(* CODESYS project Uppgift-13.project

Project tree, tasks and I/O mapping:
  Device : CODESYS Control Win V3, 3S - Smart Software Solutions GmbH, order no. 305021, version 3.5.10.40
    application Application
      libraries: Standard, * (System)
      task MainTask (cyclic, interval t#20ms, priority 1) calls PLC_PRG
      program PLC_PRG [SFC]: OpenDoor, ClosingDoor, HooldDoor, HoldLampLight, ResetValues
      global variables GVL
      Symbols
*)

// Device/Application/GVL
{attribute 'qualified_only'}
VAR_GLOBAL
	PushButton: BOOL;
	SensorOpen: BOOL;
	SensorClose: BOOL;
	MotorForward: BOOL;
	MotorReverse: BOOL;
	TopLight: BOOL;
	DOOROPENLOCK: BOOL; // Is used for lock the door open.
	HoldDoorTime: TON;
END_VAR

// Device/Application/PLC_PRG
PROGRAM PLC_PRG
VAR
	HoldDoorTime: TON;
	DoorHoldTimeElipse: TIME;
	DoorHoldTimeElipse2: TIME;
	HoldDoorTimeOff: TOF;
	TON_0: TON;
	TOF_0: TOF;
	Lampsignal: BOOL;
	BlinkingLampsignal: BOOL;
END_VAR
VAR // added by the converter: edge detectors and wires of the graphical bodies
    _w1, _w2, _w3, _w4 : ANY;
END_VAR

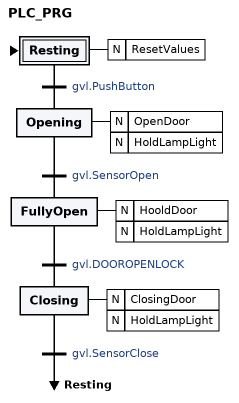
INITIAL_STEP Resting:
    ResetValues(N);
END_STEP
TRANSITION FROM Resting TO Opening
    := gvl.PushButton;
END_TRANSITION
STEP Opening:
    OpenDoor(N);
    HoldLampLight(N);
END_STEP
TRANSITION FROM Opening TO FullyOpen
    := gvl.SensorOpen;
END_TRANSITION
STEP FullyOpen:
    HooldDoor(N);
    HoldLampLight(N);
END_STEP
TRANSITION FROM FullyOpen TO Closing
    := gvl.DOOROPENLOCK;
END_TRANSITION
STEP Closing:
    ClosingDoor(N);
    HoldLampLight(N);
END_STEP
TRANSITION FROM Closing TO Resting
    := gvl.SensorClose;
END_TRANSITION

ACTION OpenDoor:
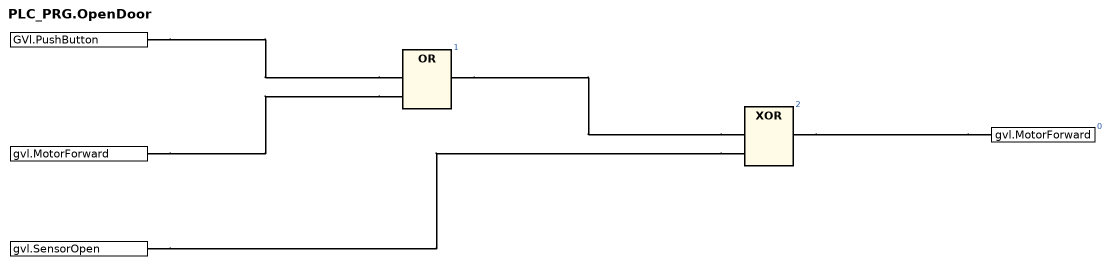
gvl.MotorForward := _w1;
_w1 := (GVl.PushButton OR gvl.MotorForward) XOR gvl.SensorOpen;
END_ACTION

ACTION ClosingDoor:
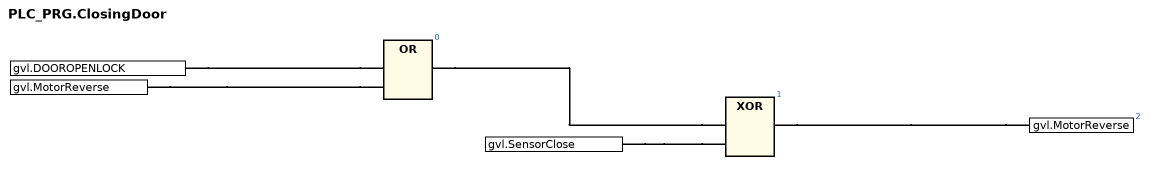
gvl.MotorReverse := (gvl.DOOROPENLOCK OR gvl.MotorReverse) XOR gvl.SensorClose;
END_ACTION

ACTION HooldDoor:
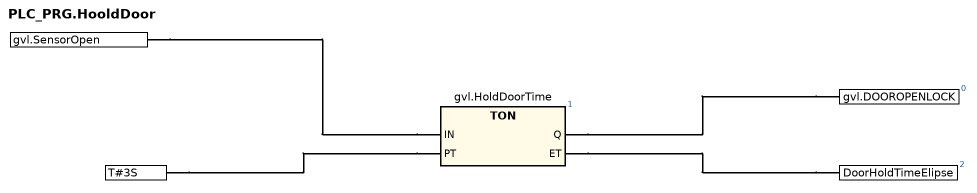
gvl.DOOROPENLOCK := gvl.HoldDoorTime.Q;
gvl.HoldDoorTime(IN := gvl.SensorOpen, PT := T#3S); // TON
DoorHoldTimeElipse := gvl.HoldDoorTime.ET;
END_ACTION

ACTION HoldLampLight:
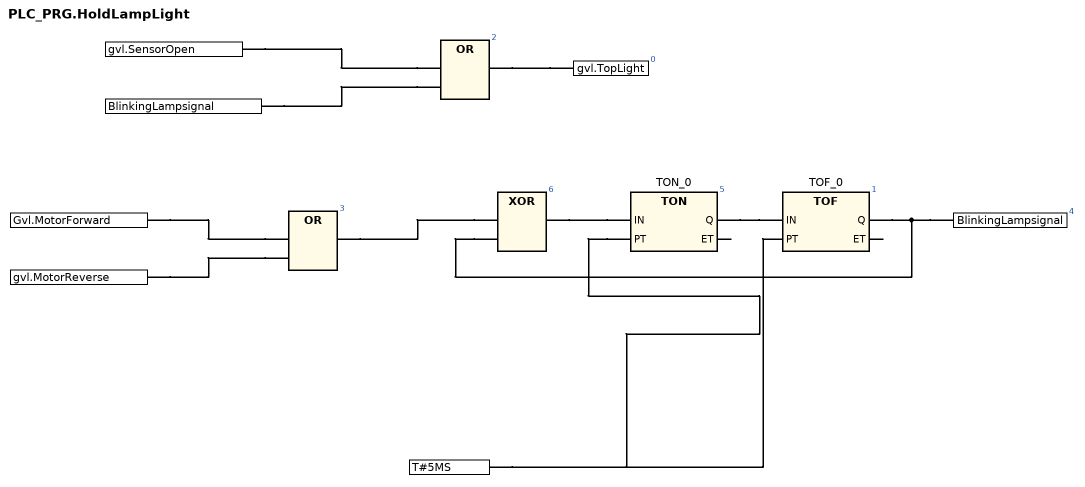
gvl.TopLight := _w2;
TOF_0(IN := TON_0.Q, PT := T#5MS); // TOF
_w2 := gvl.SensorOpen OR BlinkingLampsignal;
_w3 := Gvl.MotorForward OR gvl.MotorReverse;
BlinkingLampsignal := TOF_0.Q;
TON_0(IN := _w4, PT := T#5MS); // TON
_w4 := _w3 XOR TOF_0.Q;
END_ACTION

ACTION ResetValues:
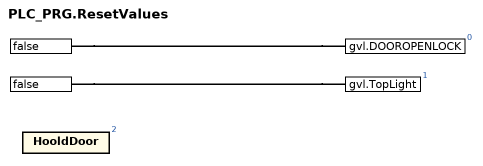
gvl.DOOROPENLOCK := false;
gvl.TopLight := false;
HooldDoor();
END_ACTION

END_PROGRAM
